(* PLC project CoDeSys External Library Template, WAGO e!COCKPIT e!COCKPIT, author 3S - Smart Software Solutions GmbH *)
(* stored: creationDateTime 2019-10-29T12:22:40.4104644, version 3.5.5.30, modificationDateTime 2019-10-24T14:40:07.960949, organization 3S - Smart Software Solutions GmbH *)
(* Library project template with all possible element types, docu and a sample project structure *)

(* values of enumPPPSLicznikCieplaMultical403Error: BrakKomunikacji: Brak komunikacji z węzłem; AlarmCzujnikaPrzeplywu: Alarm braku zmiany wartości czujnika przepływu; AlarmCzujnikaZasilania: Alarm braku zmiany wartości czujnika temp. zasilania; AlarmCzujnikaPowrotu: Alarm braku zmiany wartości czujnika temp. powrotu *)

(* Autor: Artur Wyszomirski, 2019-08-07-AWy Prawa majątkowe: Solwena Sp. z o.o., Aktualizacje: Opis: Enumeracja alarmów w fb licznia ciepła Multical403 *)
{attribute 'qualified_only'}
{attribute 'strict'}
TYPE enumPPPSLicznikCieplaMultical403Error : (BrakKomunikacji := 1, AlarmCzujnikaPrzeplywu := 2, AlarmCzujnikaZasilania := 3, AlarmCzujnikaPowrotu := 4);
END_TYPE
